// TwinCAT 3 PLC project MainPLCProject
// ProgramVersion: 3.1.4024.0
// libraries:
//   Tc2_Standard, * (Beckhoff Automation GmbH)
//   Tc2_System, * (Beckhoff Automation GmbH)
//   Tc2_TcpIp, * (Beckhoff Automation GmbH)
//   Tc2_Utilities, * (Beckhoff Automation GmbH)
//   Tc3_Module, * (Beckhoff Automation GmbH)
//   VisuDialogs, * (System)
//   VisuSymbols,3.5.10.0,System
// project tree:
//   DUTs/ ArmMovementState.TcDUT, ClientState.TcDUT, Command.TcDUT, COM_MODE.TcDUT, DataExchangeState.TcDUT, Message.TcDUT, MessageLogData.TcDUT, ReceiveStatus.TcDUT, SendStatus.TcDUT
//   DUTs/Robot Structs/ Joint.TcDUT, Position.TcDUT, RobotData.TcDUT, Timer.TcDUT
//   / GlobalTextList.TcGTLO, PlcTask.TcTTO, Visualization Manager.TcVMO (not stored)
//   GVLs/ GVL.TcGVL, GVL_Constants.TcGVL, GVL_RobotArmConstants.TcGVL
//   POUs/Classes/ ArmMovementHandler.TcPOU, COMMUNICATION.TcPOU, MESSAGE_CREATOR.TcPOU, MESSAGE_HANDLER.TcPOU, ROBOT_DATA_HANDLER.TcPOU, TCPClient.TcPOU
//   POUs/Helpers/ AddCounterToMessage.TcPOU, LogToWarning.TcPOU, ShiftHistoryLeft.TcPOU
//   POUs/InverseKinematics/ GetAngleDegreesFrom3Sides.TcPOU, GetAngleDegreesFromOppositeAndAdjacent.TcPOU, GetArm1AndArm2Degrees.TcPOU, GetArm3RotationPerpendicularToGround.TcPOU, GetBaseAngleDegrees.TcPOU, GetDistanceToPositionFromBase2D.TcPOU, GetHypotenuse.TcPOU, GetXSide.TcPOU, GetZSide.TcPOU, RadiansToDegrees.TcPOU
//   POUs/ MAIN.TcPOU
//   VISUs/ VisualizationControlPanel.TcVIS
// real-time tasks:
//   TASK PlcTask: cycle T#10ms, priority 20, ADS port 350
//   TASK HeartbeatTask: cycle T#50000us, priority 1, ADS port 351

CONFIGURATION MainPLCProject
    RESOURCE PLC ON TwinCAT3
        TASK PlcTask(INTERVAL := T#10ms, PRIORITY := 20);
        PROGRAM MAIN WITH PlcTask : MAIN;
    END_RESOURCE
END_CONFIGURATION

// ---- DUTs/ArmMovementState.TcDUT
{attribute 'qualified_only'}
{attribute 'strict'}
TYPE ArmMovementState :
(
	NONE,
	IDLE,
	PICKING,
	DROPPING
);
END_TYPE

// ---- DUTs/ClientState.TcDUT
{attribute 'qualified_only'}
{attribute 'strict'}
TYPE ClientState :
(
	IDLE,
	SENDING,
	RECEIVING
) := IDLE;
END_TYPE

// ---- DUTs/Command.TcDUT
TYPE Command :
STRUCT CONSTANT
	Start : STRING(9) := 'CRISTART';
	End : STRING(7) := 'CRIEND';
	MovementVar : STRING(4) := 'VAR';
	Heartbeat : STRING(9) := 'ALIVEJOG';
	
END_STRUCT
END_TYPE

// ---- DUTs/COM_MODE.TcDUT
{attribute 'qualified_only'}
{attribute 'strict'}
TYPE COM_MODE :
(
	Robot,
	Monarco
);
END_TYPE

// ---- DUTs/DataExchangeState.TcDUT
{attribute 'qualified_only'}
{attribute 'strict'}
TYPE DataExchangeState :
(
	IDLE,
	START,
	WORKING,
	ERROR
) := START;
END_TYPE

// ---- DUTs/Message.TcDUT
// Pre-made robot messages
TYPE Message :
STRUCT CONSTANT
	Connect : STRING(30) := 'CMD Connect';
	AliveDemo : STRING(63) := 'ALIVEJOG 40.0 50.0 40.0 30.0 30.0 0.0 0.0 0.0 0.0';	//Do not use, only for testing!
	EnableMessage : STRING(80) := 'CMD Enable';
END_STRUCT
END_TYPE

// ---- DUTs/MessageLogData.TcDUT
TYPE MessageLogData :
STRUCT
	systemTimeString : T_MaxString := '';
	message : STRING(GVL_Constants.MAX_RECEIVE_MESSAGE_LENGTH) := '';
END_STRUCT
END_TYPE

// ---- DUTs/ReceiveStatus.TcDUT
{attribute 'qualified_only'}
{attribute 'strict'}
TYPE ReceiveStatus :
(
	WAITING,
	RECEIVING,
	DONE,
	FAIL,
	TIMEOUT
) := RECEIVING;
END_TYPE

// ---- DUTs/Robot Structs/Joint.TcDUT
TYPE Joint :
STRUCT
	curPosition : LREAL;
	curSpeed : LREAL;
	setSpeed : LREAL;
	timer : TIMER;
END_STRUCT
END_TYPE

// ---- DUTs/Robot Structs/Position.TcDUT
TYPE Position :
STRUCT
	x : LREAL;	//Depth
	z : LREAL;	//Width
	y : LREAL;	//Height
END_STRUCT
END_TYPE

// ---- DUTs/Robot Structs/RobotData.TcDUT
TYPE RobotData :
STRUCT
	//Variables will be manipulated by Unity via ADS
	targetX : LREAL;
	targetY : LREAL;
	targetZ : LREAL;	
	isBusy : ARRAY[0..4] OF BOOL;	//Global value for all joints
	
	hasNewData : BOOL := FALSE;
	isAtDefaultPosition : BOOL := FALSE;	
	isAtDefaultPositionInt : INT := 0;		
	hasPickedUp : INT	:= 0;
	
	joint0 : Joint;
	joint1 : Joint;
	joint2 : Joint;
	joint3 : Joint;
	joint4 : Joint;
	
	
END_STRUCT
END_TYPE

// ---- DUTs/Robot Structs/Timer.TcDUT
TYPE Timer :
STRUCT
	timerTime : TIME;
	timerStart : BOOL;
	timerCon : TON;
END_STRUCT
END_TYPE

// ---- DUTs/SendStatus.TcDUT
{attribute 'qualified_only'}
{attribute 'strict'}
TYPE SendStatus :
(
	SENDING,
	FAIL,
	SUCCESS
) := SENDING;
END_TYPE

// ---- GVLs/GVL.TcGVL
{attribute 'qualified_only'}
VAR_GLOBAL
	// COMMUNICATION variables
	ReceivedStringArray : ARRAY[0..200] OF STRING;
	ReceivedStringWordCounter : INT := 0;

	ReceivedCMD : STRING := '';
	VarValue : STRING := '';
	VarType : STRING := '';
	VarName : STRING := '';
	//
	
	robotData : RobotData;
END_VAR

// ---- GVLs/GVL_Constants.TcGVL
{attribute 'qualified_only'}
VAR_GLOBAL CONSTANT
	MAX_RECEIVE_MESSAGE_LENGTH : UDINT := 2048;
	MAX_HISTORY_SIZE : BYTE := 10;
END_VAR

// ---- GVLs/GVL_RobotArmConstants.TcGVL
{attribute 'qualified_only'}
VAR_GLOBAL CONSTANT
	//All robot values are in mm
	PICKUP_AREA_DEPTH : LREAL := 60.0 * 10;
	PICKUP_AREA_WIDTH : LREAL := 60.0 * 10;
	
	//Values in mm
	DISTANCE_TO_PICKUP_AREA : LREAL := 90.0;	//Real: 90mm
	ARM_BASE_HEIGHT : LREAL := 310;
	GRABBER_HEIGHT : LREAL := 0.0;
	ARM_1_LENGTH : LREAL := 340.0;
	ARM_2_LENGTH : LREAL := 265.0;
	ARM_3_LENGTH : LREAL := 170.0;
	Pi : LREAL := 3.141592653589793238463;
	
	DROPOFF_X : LREAL := 450.0;	//MM	//TODO: Use DEPTH/2
	DROPOFF_Z : LREAL := PICKUP_AREA_WIDTH / 2;	//MM
	//Height is taken from the pickedup target
	DROPOFF_BASE_OFFSET : LREAL := -90.0;	//Degrees
	

	
	//Values in degrees
	MAXIMUM_BASE_ROTATION_FROM_CENTER : LREAL := 120.0;
	
END_VAR

// ---- POUs/MAIN.TcPOU
PROGRAM MAIN
VAR CONSTANT
	LOCAL_IP : T_IPv4Addr := '127.0.0.1';
	LOCAL_PORT : UDINT := 8080;

	REMOTE_IP : T_IPv4Addr := '192.168.3.1';
	REMOTE_PORT : UDINT := 8080;
	
	ROBOT_IP : T_IPv4Addr := '192.168.3.11';
	ROBOT_PORT : UDINT := 3920;
	
	MONARCO_IP : T_IPv4Addr := '192.168.3.125';
	MONARCO_PORT : UDINT := 8080;
	//TODO: Remove? not used anywhere afaik
	command : Command := ();
	message : Message := ();

	testPosition : Position := (x := 250.0, z := 250.0, y := 250.0);
	
END_VAR
VAR
	isSetUp : BOOL := FALSE;	

	buttonConnectPressed : BOOL;
	buttonDisconnectPressed : BOOL;	
	buttonSendPressed : BOOL;
	buttonConnectToRobotPressed : BOOL;
	buttonDebugSendPressed : BOOL;
	buttonEnableMotorsPressed : BOOL;
	buttonDisableMotorsPressed : BOOL;
	buttonLeft0Pressed : BOOL;
	buttonRight0Pressed : BOOL;
	buttonLeft1Pressed : BOOL;
	buttonRight1Pressed : BOOL;
	buttonLeft2Pressed : BOOL;
	buttonRight2Pressed : BOOL;
	buttonLeft3Pressed : BOOL;
	buttonRight3Pressed : BOOL;
	buttonStopPressed : BOOL;
	
	connectTrigger : R_TRIG;
	disconnectTrigger : R_TRIG;
	sendTrigger : R_TRIG;
	connectToRobotTrigger : R_TRIG;
	debugSendTrigger : R_TRIG;
	enableMotorsTrigger : R_TRIG;
	disableMotorsTrigger : R_TRIG;
	stopTrigger : R_TRIG;
	right0Trigger : R_TRIG;
	left0Trigger : R_TRIG;
	right1Trigger : R_TRIG;
	left1Trigger : R_TRIG;
	right2Trigger : R_TRIG;
	left2Trigger : R_TRIG;
	right3Trigger : R_TRIG;
	left3Trigger : R_TRIG;
	
	client : TCPClient(MONARCO_IP, MONARCO_PORT, isEnabled := FALSE);	//Note: make sure the COM_MODE is set properly, as it overwrites these values
	LocalSystemTime : FB_LocalSystemTime;
	
	// COMMUNICATION message handling
	MessageBase : COMMUNICATION(CommunicationMODE := COM_MODE.Robot); // change this to switch between robot and monarco mode!!
	messageHandler : MESSAGE_HANDLER();
	MessageERROR : int := 0;
	//
	// ROBOT_DATA handling
	RobotDataHandler : ROBOT_DATA_HANDLER;
	armMovementHandler : ArmMovementHandler;
	//
	
	connectionMessage : STRING(20) := 'Disconnected';
	isHeartbeatEnabled : BOOL := FALSE;
	
	closeAllConnections : FB_SocketCloseALL();
	closeAll : BOOL := TRUE;	//Close all on initial startup
	
	//messageToServer : T_MaxString := 'CRISTART 1 CMD Connect CRIEND';
	messageToServer : T_MaxString := 'Hello world 2.0 CRIEND';
	debugMessageToServer : T_MaxString := 'VAR Joint 0.0 0.0 0.0 0.0 0.0 0.0 0.0 0.0 0.0';
	messageFromServer : STRING(GVL_Constants.MAX_RECEIVE_MESSAGE_LENGTH) := '';
	//finalSendMsg : STRING(100);
	
	heartbeatTimer : TON;
	heartbeatInterval : TIME := T#100MS;
	
	sendCounter : INT := 1;
	finalAliveMessage : STRING(100) := '';
	totalMessagesFromServerCount : UDINT := 0;
	
	currentTime : TIMESTRUCT;
	messageHistoryArray : ARRAY [0.. GVL_Constants.MAX_HISTORY_SIZE - 1] OF MessageLogData;
	currentHistoryIndex : BYTE := 0;
	currentMessageLogData : MessageLogData;
	
	//Testing
	dummyHeartbeatValues : STRING(80);
	dummyMoveValues : STRING(80);
	

END_VAR

//On PLC reset/program download, close all connections
HandlePLCReset();

HandleSetup();
// === ===

// === UI Handling ===
HandleUI();

// === Message Sending ===
HandleMessageSending();

// === Message Handling ===
HandleMessageReceiving();

// === Heartbeat ===
HandleHeartbeat();

// === Arm movement ===
armMovementHandler();

// === Socket client ====
client(totalMessagesReceived => totalMessagesFromServerCount);



IF (GVL.robotData.isAtDefaultPosition = TRUE) THEN
	GVL.robotData.isAtDefaultPositionInt := 1;
ELSE
	GVL.robotData.isAtDefaultPositionInt := 0;
	
END_IF

METHOD PRIVATE HandleHeartbeat : BOOL
VAR_INPUT
END_VAR
heartbeatTimer(IN := isHeartbeatEnabled, PT := heartbeatInterval);

IF (heartbeatTimer.Q AND client.IsClientEnabled) THEN
	heartbeatTimer(IN := FALSE);
	// Send all movement data to the robot via the hardbeat.
	client.Send(messageToSend := MessageBase.CREATE('ALIVEJOG', RobotDataHandler.DATA_TO_STRING(), ERROR => MessageERROR));
END_IF
END_METHOD

METHOD PRIVATE HandleMessageReceiving : BOOL
VAR_INPUT
END_VAR
IF (client.NewMessageAvailable(clearFlag := TRUE)) THEN
	//Update history
	IF (currentHistoryIndex >= GVL_Constants.MAX_HISTORY_SIZE) THEN
		//Ran out of history space, discard youngest member
		currentHistoryIndex := GVL_Constants.MAX_HISTORY_SIZE;
		ShiftHistoryLeft(arr := messageHistoryArray);
	ELSE
		//Can still append
		currentHistoryIndex := currentHistoryIndex + 1;
	END_IF
	
	//Handle message
	MessageBase.HANDLE(messageFromServer);
	
	//Add new entry
	currentMessageLogData.message := messageFromServer;	
	currentMessageLogData.systemTimeString := SYSTEMTIME_TO_STRING(in := currentTime);
	messageHistoryArray[currentHistoryIndex - 1] := currentMessageLogData;
END_IF
END_METHOD

METHOD PRIVATE HandleMessageSending : BOOL
VAR_INPUT
END_VAR
CASE MessageBase.COMMUNICATION_MODE OF
	COM_MODE.Robot:
// ROBOT COM
		IF (sendTrigger.Q) THEN  // debug: send move command to robot.
			//TODO: Rework to use +- buttons (like in the C# application)
//			client.Send(messageToSend := MessageBase.CREATE(COMMAND := 'VAR', COMMAND_DETAILS := 'GetPosVariable Joint', ERROR => MessageERROR));
//			RobotDataHandler.DEGREES_TO_MOVEMENT_DATA(degrees := -45, jointNr := 0);
//			RobotDataHandler.DEGREES_TO_MOVEMENT_DATA(degrees := -34.8529, jointNr := 1);
//			RobotDataHandler.DEGREES_TO_MOVEMENT_DATA(degrees := -18.5157, jointNr := 2);
//			RobotDataHandler.DEGREES_TO_MOVEMENT_DATA(degrees := 53.3685, jointNr := 3);
			//RobotDataHandler.SET_JOINTS_TO_POSITION(X := 250.0, Z:= 250.0, Y := 250.0, baseOffsetDegrees := 0.0);
			
			GVL.robotData.targetX := 253.0;
			GVL.robotData.targetZ := 171.0;
			GVL.robotData.targetY := 160.0;
			
			GVL.robotData.hasNewData := TRUE;
		END_IF

		IF (debugSendTrigger.Q) THEN // debug: not in use yet.
//			client.Send(messageToSend := MessageBase.CREATE(COMMAND := 'CMD', COMMAND_DETAILS := 'Reset', ERROR => MessageERROR));
			RobotDataHandler.DEGREES_TO_MOVEMENT_DATA(degrees := 0, jointNr := 0);
			RobotDataHandler.DEGREES_TO_MOVEMENT_DATA(degrees := 0, jointNr := 1);
			RobotDataHandler.DEGREES_TO_MOVEMENT_DATA(degrees := 0, jointNr := 2);
			RobotDataHandler.DEGREES_TO_MOVEMENT_DATA(degrees := 0, jointNr := 3);
		END_IF
		
		IF (left0Trigger.Q) THEN  // debug: send move command to robot.
			GVL.robotData.joint0.curSpeed := 20.0;
		END_IF
		
		IF (right0Trigger.Q) THEN 
			
			GVL.robotData.joint0.curSpeed := -20.0;
		END_IF
		
		IF (left1Trigger.Q) THEN  // debug: send move command to robot.
			GVL.robotData.joint1.curSpeed := 20.0;
		END_IF
		
		IF (right1Trigger.Q) THEN 
			
			GVL.robotData.joint1.curSpeed := -20.0;
		END_IF
		
		IF (left2Trigger.Q) THEN  // debug: send move command to robot.
			GVL.robotData.joint2.curSpeed := 20.0;
		END_IF
		
		IF (right2Trigger.Q) THEN 
			
			GVL.robotData.joint2.curSpeed := -20.0;
		END_IF
		
		IF (left3Trigger.Q) THEN  // debug: send move command to robot.
			GVL.robotData.joint3.curSpeed := 20.0;
		END_IF
		
		IF (right3Trigger.Q) THEN 
			
			GVL.robotData.joint3.curSpeed := -20.0;
		END_IF
		
		IF (stopTrigger.Q) THEN 
			GVL.robotData.joint0.curSpeed := 0.0;
			GVL.robotData.joint1.curSpeed := 0.0;
			GVL.robotData.joint2.curSpeed := 0.0;
			GVL.robotData.joint3.curSpeed := 0.0;
		END_IF

		IF (connectToRobotTrigger.Q) THEN
			client.Send(messageToSend := MessageBase.CREATE(COMMAND := 'CMD', COMMAND_DETAILS := 'Connect', ERROR => MessageERROR));
			isHeartbeatEnabled := TRUE;
		END_IF

		IF (enableMotorsTrigger.Q) THEN
			client.Send(messageToSend := MessageBase.CREATE(COMMAND := 'CMD', COMMAND_DETAILS := 'Enable', ERROR => MessageERROR));
		END_IF
		
		IF (disableMotorsTrigger.Q) THEN
			client.Send(messageToSend := MessageBase.CREATE(COMMAND := 'CMD', COMMAND_DETAILS := 'Disable', ERROR => MessageERROR));
		END_IF
//		
	COM_MODE.Monarco:
// MONARCO COM
		IF (sendTrigger.Q) THEN 
			client.Send(messageToSend := MessageBase.CREATE(COMMAND := 'CMD', COMMAND_DETAILS := 'LED_ON', ERROR => MessageERROR));
		END_IF

		IF (debugSendTrigger.Q) THEN
			client.Send(messageToSend := MessageBase.CREATE(COMMAND := 'CMD', COMMAND_DETAILS := 'LED_OFF', ERROR => MessageERROR));
		END_IF
//
END_CASE
END_METHOD

METHOD HandlePLCReset : BOOL
VAR_INPUT
END_VAR
IF (closeAll) THEN	
	closeAll := FALSE;
	closeAllConnections(sSrvNetId := '', bExecute := TRUE, tTimeout := T#10S);
ELSE
	closeAllConnections(bExecute := FALSE);
END_IF

IF (closeAllConnections.bBusy) THEN
	RETURN;	//Do not continue the program until all connections are closed
END_IF
END_METHOD

METHOD HandleSetup : BOOL
VAR_INPUT
END_VAR
IF (NOT isSetUp) THEN
	armMovementHandler.BindRobotDataHandler(dataHandler := RobotDataHandler);

	isSetUp := TRUE;
END_IF
END_METHOD

METHOD HandleUI : BOOL
VAR_INPUT
END_VAR
LocalSystemTime(bEnable := TRUE, tTimeout := T#1S, systemTime => currentTime);

connectTrigger(CLK := buttonConnectPressed);
disconnectTrigger(CLK := buttonDisconnectPressed);
sendTrigger(CLK := buttonSendPressed);
connectToRobotTrigger(CLK := buttonConnectToRobotPressed);
debugSendTrigger(CLK := buttonDebugSendPressed);
enableMotorsTrigger(CLK := buttonEnableMotorsPressed);
disableMotorsTrigger(CLK := buttonDisableMotorsPressed);
left0Trigger(CLK := buttonLeft0Pressed);
right0Trigger(CLK := buttonRight0Pressed);
left1Trigger(CLK := buttonLeft1Pressed);
right1Trigger(CLK := buttonRight1Pressed);
left2Trigger(CLK := buttonLeft2Pressed);
right2Trigger(CLK := buttonRight2Pressed);
left3Trigger(CLK := buttonLeft3Pressed);
right3Trigger(CLK := buttonRight3Pressed);
stopTrigger(CLK := buttonStopPressed);

IF (client.IsConnected) THEN
	connectionMessage := 'Connected';
ELSE
	connectionMessage := 'Disconnected';
END_IF

IF (connectTrigger.Q) THEN
	//Note: Not sure if this is a good idea, as it is burried in the code and can lead to unexpected behaviour
	CASE MessageBase.COMMUNICATION_MODE OF
	// check for communication mode and set IP for this mode.
		COM_MODE.Robot:
			client.RemoteServerAddress := ROBOT_IP;
			client.RemoteServerPort := ROBOT_PORT;
		
		COM_MODE.Monarco:
			client.RemoteServerAddress := MONARCO_IP;
			client.RemoteServerPort := MONARCO_PORT;
	END_CASE
	client.BindReceiveMessage(variableToBind := messageFromServer);
	client.Enable();
END_IF

IF (disconnectTrigger.Q) THEN
	client.Disable();
END_IF
END_METHOD

END_PROGRAM

// ---- POUs/Classes/TCPClient.TcPOU
FUNCTION_BLOCK TCPClient
VAR CONSTANT
	CLIENT_RECONNECT_TIME : TIME := T#31S;
	MAX_MESSAGE_LENGTH : INT := 255;
	MAX_RECEIVE_MESSAGE_LENGTH : UDINT := GVL_Constants.MAX_RECEIVE_MESSAGE_LENGTH;
END_VAR
VAR_OUTPUT
	totalMessagesReceived : UDINT := 0;
END_VAR
VAR
	m_isClientEnabled : BOOL := TRUE;	
	m_serverNetID : STRING(80) := '';
	
	ClientServerConnection : FB_ClientServerConnection;
	SocketSend : FB_SocketSend;
	SocketReceive : FB_SocketReceive;
	//m_clientDataExchanger : ClientDataExchanger;	//Note implemented yet: leave for later, use as
	m_socketHandle : T_HSOCKET;
	
	
	m_remoteServerAddress : T_IPv4Addr;	
	m_remoteServerPort : UDINT := 0;
	
	//Note: make it an input and send only when the class is called?
	m_messageToSend : T_MaxString := 'Hello world!';
	//m_messageReceived : T_MaxString;	// The latest message received from the server //TODO: REMOVE, Depricated
	m_messageReceivedRef : REFERENCE TO STRING(MAX_RECEIVE_MESSAGE_LENGTH);
	
	m_isConnected : BOOL := FALSE;
	m_isBusy : BOOL;
	m_errorOccured : BOOL;
	m_lastErrorId : UDINT;
	
	
	m_currentSocketState : Tc2_TcpIp.E_SocketConnectionState;
	m_currentState : ClientState := ClientState.RECEIVING;	

	m_sendDataExchangeState : DataExchangeState := DataExchangeState.START;	
	m_sendRequested: BOOL;
	m_sendStatus : SendStatus;
	m_sendErrorId : UDINT;
	m_sendTimeout : TIME := T#15S;	//Note: Lower?
	//m_sendTimeout : TIME := T#1M;	//Note: Lower?
	
	//Receiving
	m_receiveDataExchangeState : DataExchangeState := DataExchangeState.IDLE;	
	m_isReceiveTimerEnabled : BOOL := TRUE;
	m_receiveTimer : TON();
	m_isReceiveTimeoutEnabled : BOOL := FALSE;	
	m_receiveTimeoutTimer : TON();
	m_receiveBuffer : STRING(MAX_RECEIVE_MESSAGE_LENGTH) := '';
	m_totalBytesReceived : UDINT := 0;
	m_receiveTimeout : TIME := T#1M;
	m_readInterval : TIME := T#10MS;
//	m_receiveMessageDelimiter : BYTE := F_ToASC(';');	//Note: Use plain 0 (without F_ToASC()) for \0
	m_receiveMessageDelimiter : BYTE := 0;	//'\0'	//Not used currently
	m_delimiterString : STRING(80) := 'CRIEND';
	m_receivedMessage : T_MaxString := '';
	m_receiveStatus : ReceiveStatus;
	m_newDataAvailable : BOOL := FALSE;	//Reset to false when it is read
	m_receiveErrorId : UDINT := 0;
	m_totalMessagesReceived : UDINT := 0;
END_VAR

//Handler code
//Does that need to be executed every cycle or can I put it in eSOCKET_DISCONNECTED state?
ClientServerConnection(sSrvNetID := m_serverNetID,
						 nMode := 0,
						 sRemoteHost := RemoteServerAddress,
						 nRemotePort := m_remoteServerPort,
						 tReconnect := CLIENT_RECONNECT_TIME,	//MAYBE
						 bEnable := IsClientEnabled,
						 bBusy => m_isBusy,
						 bError => m_errorOccured,
						 nErrId => m_lastErrorId,
						 hSocket => m_socketHandle,
						 eState => m_currentSocketState);

CASE m_currentSocketState OF
	E_SocketConnectionState.eSOCKET_DISCONNECTED:
		m_isConnected := FALSE;
	//
	E_SocketConnectionState.eSOCKET_SUSPENDED:
	//Change from disconnected to connected or vise versa
		m_isConnected := FALSE;
	//
	E_SocketConnectionState.eSOCKET_CONNECTED:
		m_isConnected := TRUE;
END_CASE

IF (NOT m_isConnected) THEN
	RETURN;
END_IF

// Executed only if a connection is established

CASE m_currentState OF
	//
	ClientState.SENDING:
		m_sendStatus := SendMessage(messageToSend := m_messageToSend, timeout := m_sendTimeout, errorId => m_sendErrorId);
		IF (m_sendStatus = SendStatus.SUCCESS) THEN
			m_currentState := ClientState.RECEIVING;
		ELSIF (m_sendStatus = SendStatus.FAIL) THEN
			//Sending failed
			ADSLOGDINT(msgCtrlMask := ADSLOG_MSGTYPE_WARN, msgFmtStr := 'Send fail error: %d', dintArg := UDINT_TO_DINT(m_sendErrorId));
			m_currentState := ClientState.RECEIVING;
		END_IF
		
	//
	ClientState.RECEIVING:
		m_receiveStatus := Receive(timeout := m_receiveTimeout, 
									readInterval := m_readInterval, 
									messageDelimiter := m_receiveMessageDelimiter,	//Currently not used
									errorId => m_receiveErrorId);
		
		IF (m_receiveStatus <> ReceiveStatus.RECEIVING) THEN
			IF (m_receiveStatus = ReceiveStatus.DONE) THEN
				//
				totalMessagesReceived := totalMessagesReceived + 1;
				m_newDataAvailable := TRUE;
			END_IF
			
			IF (m_receiveStatus = ReceiveStatus.FAIL) THEN
				//Fail Handling
				//How does it get to error and the error is 0??
				LogToWarning(msgFmtStr := 'Receive fail error: %s', messageArg := UDINT_TO_STRING(m_receiveErrorId));
			END_IF
			
			IF (m_receiveStatus = ReceiveStatus.TIMEOUT) THEN
				//Timeout handling
				LogToWarning(msgFmtStr := 'Receive timed out', messageArg := '');
				//Disable();	//Disable on timeout
			END_IF
	
			IF (m_sendRequested) THEN
				m_sendRequested := FALSE;
				m_sendErrorId := 0;
				m_currentState := ClientState.SENDING;
			END_IF
		END_IF						
	
	// After done receiving, go to idle?
	//
END_CASE

METHOD PUBLIC BindReceiveMessage : BOOL
VAR_INPUT
	variableToBind : REFERENCE TO STRING(MAX_RECEIVE_MESSAGE_LENGTH);
END_VAR
m_messageReceivedRef REF= variableToBind;
END_METHOD

METHOD PUBLIC Disable : BOOL
m_isClientEnabled := False;
END_METHOD

METHOD PUBLIC Enable : BOOL
VAR_INPUT
END_VAR
m_isClientEnabled := TRUE;
END_METHOD

METHOD FB_init : BOOL
VAR_INPUT
	bInitRetains : BOOL; // if TRUE, the retain variables are initialized (warm start / cold start)
	bInCopyCode : BOOL;  // if TRUE, the instance afterwards gets moved into the copy code (online change)
	
	remoteServerAddress : T_IPv4Addr := '127.0.0.1';
	remoteServerPort : UDINT := 8080;
	isEnabled : BOOL := FALSE;
END_VAR
m_remoteServerAddress := remoteServerAddress;
m_remoteServerPort := remoteServerPort;
m_isClientEnabled := isEnabled;
END_METHOD

PROPERTY IsClientEnabled : BOOL
GET
IsClientEnabled := m_isClientEnabled;
END_GET
END_PROPERTY

PROPERTY IsConnected : BOOL
GET
IsConnected := m_isConnected;
END_GET
END_PROPERTY

PROPERTY LastSendStatus : SendStatus
GET
LastSendStatus := m_sendStatus;
END_GET
END_PROPERTY

METHOD PUBLIC NewMessageAvailable : BOOL
VAR_INPUT
	clearFlag : BOOL := FALSE;	//Clears the new message flag if set to true, does not otherwise
END_VAR
NewMessageAvailable := m_newDataAvailable;

IF (clearFLag) THEN
	m_newDataAvailable := FALSE;
END_IF
END_METHOD

METHOD PRIVATE Receive : ReceiveStatus
VAR_INPUT
	timeout : TIME;// := T#10S;
	readInterval : TIME := T#10MS;
	messageDelimiter : BYTE := 0;
END_VAR

VAR_OUTPUT
	errorId : UDINT;
END_VAR

VAR
	errorOccurred : BOOL;	//can sty
	isBusy : BOOL;	//can stay																
	
	timedout : BOOL := FALSE;	//Output of TON
	receivedBytes : UDINT := 0;	//Output, should be fine to be here
	
	startPosition : UDINT := 0;	//Can stay, assigned before used
	endPosition : UDINT := 0;	//Can stay, assigned before used
	currentFrameLength : UDINT := 0; // Length of string received this cycle	//Should be fine
	posOfDelimiter : UDINT := 0;
	
	
	index : UDINT := 0;	//For-loop index
	
END_VAR
m_receiveTimer(IN := m_isReceiveTimerEnabled);
m_receiveTimeoutTimer(IN := m_isReceiveTimeoutEnabled, PT := timeout, Q => timedout);

CASE m_receiveDataExchangeState OF
	DataExchangeState.IDLE:
		//Reset variables
		m_isReceiveTimerEnabled := FALSE;
		m_receiveTimer(IN := m_isReceiveTimerEnabled, PT := T#0MS); 	//Do not wait for the first read
		m_isReceiveTimeoutEnabled := FALSE;
		Receive := ReceiveStatus.WAITING;
		m_receiveDataExchangeState := DataExchangeState.START;
	//
	DataExchangeState.START:
		Receive := ReceiveStatus.WAITING;
		m_isReceiveTimerEnabled := TRUE;
		IF (m_receiveTimer.Q) THEN
			SocketReceive(bExecute := FALSE);
			SocketReceive(sSrvNetId := m_serverNetID,
						  hSocket := m_socketHandle,
						  pDest := ADR(m_receiveBuffer) + m_totalBytesReceived,
						  cbLen := SIZEOF(m_receiveBuffer) - m_totalBytesReceived,
						  tTimeout := timeout,
						  bExecute := TRUE);	
			
			m_receiveDataExchangeState := DataExchangeState.WORKING;
		END_IF
	//
	DataExchangeState.WORKING:
		Receive := ReceiveStatus.RECEIVING;
		SocketReceive(bExecute := FALSE,
				tTimeout := timeout,
				bBusy => isBusy,
				bError => errorOccurred,
				nErrId => errorId,
				nRecBytes => receivedBytes);
		//Enable timeout
		IF (NOT isBusy AND NOT errorOccurred) THEN
			IF (receivedBytes > 0) THEN
				startPosition := m_totalBytesReceived;
				//Calculate new total
				m_totalBytesReceived := m_totalBytesReceived + receivedBytes;
				endPosition := m_totalBytesReceived - 1;
				currentFrameLength := 0;
				//Only proceed if we have enough space
				IF (m_totalBytesReceived < SIZEOF(m_messageReceivedRef)) THEN
					m_receiveTimer (PT := T#0MS); //Read asap
					//Bytes received, disable timeout check
					m_isReceiveTimeoutEnabled := FALSE;
					//Search for end of message delimiter
					
					posOfDelimiter := INT_TO_UDINT(FIND(STR1 := m_receiveBuffer, STR2 := m_delimiterString));
					
					IF (posOfDelimiter = 0) THEN
						//Delimiter not found
						LogToWarning('Delim not found', '');
						RETURN;
					END_IF
					
					currentFrameLength := posOfDelimiter + 6(*delimiter size*);
					//reset dest
					m_messageReceivedRef := '';
					MEMCPY(destAddr := ADR(m_messageReceivedRef), srcAddr := ADR(m_receiveBuffer), n := currentFrameLength);
					MEMSET(destAddr := ADR(m_receiveBuffer), fillByte := 0, n := SIZEOF(m_receiveBuffer));	//Clear buffer
					m_totalBytesReceived := 0;
					
					//All received
					Receive := ReceiveStatus.DONE;
					m_receiveDataExchangeState := DataExchangeState.IDLE;
					(*
					//OLD Find TODO: Find a way to implement via a function? So that you can use both
					FOR index := startPosition TO endPosition BY 1 DO
						IF (m_receiveBuffer[index] = messageDelimiter) THEN	//End of message check
							//End of message received
							currentFrameLength := index + 1;
							
							MEMCPY(destAddr := ADR(m_messageReceivedRef), srcAddr := ADR(m_receiveBuffer), n := currentFrameLength);
							//Move the remaining data bytes to the begining
							MEMMOVE(ADR(m_receiveBuffer), ADR(m_receiveBuffer[currentFrameLength]), m_totalBytesReceived - currentFrameLength); 
							//Recalculate remaining data byte length
							m_totalBytesReceived := m_totalBytesReceived - currentFrameLength;
							//All received
							Receive := ReceiveStatus.DONE;
							m_receiveDataExchangeState := DataExchangeState.IDLE;
							EXIT;
						END_IF
					END_FOR
					*)
				ELSE	
					//No more space in the receive object
					Receive := ReceiveStatus.FAIL;
					errorId := 42;
					//LogToWarning('totalBytesReceived exceeded limit: Received: %s', UDINT_TO_STRING(receivedBytes));
					m_receiveDataExchangeState := DataExchangeState.ERROR;
				END_IF //IF (totalBytesReceived < SIZEOF(receivedMessage))
			ELSE
				//No bytes received
				m_receiveTimer (PT := readInterval);
				m_isReceiveTimeoutEnabled := TRUE;
				
				//IF (timedout) THEN
				IF (m_receiveTimeoutTimer.Q) THEN
					Receive := ReceiveStatus.TIMEOUT;
					m_receiveDataExchangeState := DataExchangeState.ERROR;
					LogToWarning('Timed out!', '');
				ELSE
					//Read again
					m_receiveDataExchangeState := DataExchangeState.START;
				END_IF
			END_IF //IF (receivedBytes > 0)
		
		ELSIF (errorOccurred) THEN
			Receive := ReceiveStatus.FAIL;
			m_receiveDataExchangeState := DataExchangeState.ERROR;
		END_IF	//IF (NOT isBusy AND NOT errorOccurred)
		
	//
	DataExchangeState.ERROR:
		//Variable resets in case of an error
		m_totalBytesReceived := 0;	//Reset counter
		m_receiveBuffer := DELETE(STR := m_receiveBuffer, POS := 1, LEN := 255);	//Reset receive buffer
		m_receiveDataExchangeState := DataExchangeState.IDLE;
	//
END_CASE
END_METHOD

//Note: After reading, NewDataAvailable returns false until new data arrives
PROPERTY ReceivedData : T_MaxString
GET
ReceivedData := m_receivedMessage;
m_newDataAvailable := FALSE;
END_GET
END_PROPERTY

PROPERTY RemoteServerAddress : T_IPv4Addr
GET
RemoteServerAddress := m_remoteServerAddress;
END_GET
SET
m_remoteServerAddress := RemoteServerAddress;
END_SET
END_PROPERTY

PROPERTY RemoteServerPort : UDINT
GET
RemoteServerPort := m_remoteServerPort;
END_GET
SET
m_remoteServerPort := RemoteServerPort;
END_SET
END_PROPERTY

METHOD Send : BOOL
VAR_INPUT
	messageToSend : T_MaxString;
END_VAR
m_sendRequested := TRUE;
m_messageToSend := messageToSend;
END_METHOD

//Wrapper for SocketSend. On error, check the errorId variable
METHOD PRIVATE SendMessage : SendStatus
VAR_INPUT
	messageToSend : T_MaxString;
	timeout : TIME;
END_VAR

VAR_OUTPUT
	errorId : UDINT := 0;
END_VAR

VAR
	errorOccurred : BOOL;	
	isBusy : BOOL;	
END_VAR
CASE m_sendDataExchangeState OF
	DataExchangeState.START:
		errorId := 0;
		
		SocketSend(sSrvNetId := m_serverNetID,
				   hSocket := m_socketHandle,
				   cbLen := INT_TO_UDINT(LEN(messageToSend) + 1),
		   		   pSrc := ADR(messageToSend),
				   tTimeout := timeout,
				   bExecute := FALSE
				   );

		m_sendDataExchangeState := DataExchangeState.WORKING;
	//
	DataExchangeState.WORKING:
		
		SocketSend(bExecute := TRUE,
				   bError => errorOccurred,
		   		   nErrId => errorId,
		   		   bBusy => isBusy);
		
		IF (NOT isBusy AND NOT errorOccurred) THEN
			SendMessage := SendStatus.SUCCESS;
			m_sendDataExchangeState := DataExchangeState.START;
		ELSIF (errorOccurred) THEN
			SendMessage := SendStatus.FAIL;
			m_sendDataExchangeState := DataExchangeState.START;
		ELSIF (isBusy) THEN
			SendMessage := SendStatus.SENDING;
		END_IF 
	//
END_CASE
END_METHOD

END_FUNCTION_BLOCK

// ---- POUs/Helpers/LogToWarning.TcPOU
FUNCTION LogToWarning : BOOL
VAR_INPUT
	msgFmtStr : T_MaxString;
	messageArg : T_MaxString;
END_VAR
VAR
END_VAR

ADSLOGSTR(msgCtrlMask := ADSLOG_MSGTYPE_WARN, msgFmtStr := msgFmtStr, strArg := messageArg);

END_FUNCTION

// ---- POUs/Classes/COMMUNICATION.TcPOU
FUNCTION_BLOCK COMMUNICATION
VAR_INPUT
	
END_VAR
VAR_OUTPUT
END_VAR
VAR
	m_COMMUNICATION_MODE : COM_MODE;
	messageCreator : MESSAGE_CREATOR('CRISTART', 'CRIEND', 1);
	messageHandler : MESSAGE_HANDLER();
END_VAR

PROPERTY PUBLIC COMMUNICATION_MODE : COM_MODE
GET
COMMUNICATION_MODE := m_COMMUNICATION_MODE;
END_GET
SET
m_COMMUNICATION_MODE := COMMUNICATION_MODE;
END_SET
END_PROPERTY

METHOD PUBLIC CREATE : STRING
VAR_INPUT
	COMMAND : STRING;
	COMMAND_DETAILS : STRING;
END_VAR
VAR_OUTPUT
	ERROR : INT := 0;
END_VAR
IF (COMMUNICATION_MODE = COM_MODE.Robot) THEN 
	// creates string for robot when in Robot mode
	CREATE := MessageCreator.ROBOT_MESSAGE(COMMAND, COMMAND_DETAILS, ERROR => ERROR);
ELSIF (COMMUNICATION_MODE = COM_MODE.Monarco) THEN 
	// creates string for monarco when in Monarco mode
	CREATE := MessageCreator.MONARCO_MESSAGE_CMD(COMMAND_DETAILS, ERROR => ERROR);
			// JUST THE CMD MONARCO MESSAGE FOR NOW!!
END_IF
END_METHOD

METHOD FB_init : BOOL
VAR_INPUT
	bInitRetains : BOOL; // if TRUE, the retain variables are initialized (warm start / cold start)
	bInCopyCode : BOOL;  // if TRUE, the instance afterwards gets moved into the copy code (online change)
	
	communicationMODE : COM_MODE;
END_VAR
COMMUNICATION_MODE := communicationMode;
END_METHOD

METHOD PUBLIC HANDLE : INT
VAR_INPUT
	FULL_STRING : STRING;
END_VAR
IF (COMMUNICATION_MODE = COM_MODE.Robot) THEN 
	// handles string from robot when in Robot mode (RECEIVE_ROBOT())
	MessageHandler.RECEIVE_ROBOT(FULL_STRING, ERROR => HANDLE);
ELSIF (COMMUNICATION_MODE = COM_MODE.Monarco) THEN 
	// handles string from monarco when in Monarco mode (RECEIVE_MONARCO())
	MessageHandler.RECEIVE_MONARCO(FULL_STRING, ERROR => HANDLE);
END_IF
END_METHOD

END_FUNCTION_BLOCK

// ---- POUs/Classes/MESSAGE_CREATOR.TcPOU
FUNCTION_BLOCK PUBLIC MESSAGE_CREATOR
VAR_INPUT
END_VAR
VAR_OUTPUT
END_VAR
VAR
	m_START_COMMAND : STRING;
	m_END_COMMAND : STRING;
	m_MESSAGE_COUNT : INT;
END_VAR

PROPERTY PUBLIC END_COMMAND : STRING
GET
END_COMMAND := m_END_COMMAND;
END_GET
SET
m_END_COMMAND := END_COMMAND;
END_SET
END_PROPERTY

METHOD FB_init : BOOL
VAR_INPUT
	bInitRetains : BOOL; // if TRUE, the retain variables are initialized (warm start / cold start)
	bInCopyCode : BOOL;  // if TRUE, the instance afterwards gets moved into the copy code (online change)
	
	STARTcommand : STRING;
	ENDcommand : STRING;
	MESSAGEcount : INT;
END_VAR
START_COMMAND := STARTcommand;
END_COMMAND := ENDcommand;
MESSAGE_COUNT := MESSAGEcount;
END_METHOD

PROPERTY PUBLIC MESSAGE_COUNT : INT
GET
MESSAGE_COUNT := m_MESSAGE_COUNT;
END_GET
SET
m_MESSAGE_COUNT := MESSAGE_COUNT;
END_SET
END_PROPERTY

METHOD PUBLIC MONARCO_MESSAGE_CMD : STRING
VAR_INPUT
	COMMAND_DETAILS : STRING;
END_VAR
VAR CONSTANT
	COMMAND : STRING := 'CMD';
	SEPARATOR : STRING := ' ';
END_VAR
VAR_OUTPUT
	ERROR : INT := 0;
END_VAR
IF (COMMAND_DETAILS <> '') THEN // if command_details is not empty, create command string.
	MONARCO_MESSAGE_CMD := 
		CONCAT(COMMAND, 
		CONCAT(SEPARATOR, 
			COMMAND_DETAILS));
			
ELSE // else return error string and error code 1.
	MONARCO_MESSAGE_CMD := 'ERROR_NoCommandDetailsGiven';
	ERROR := 1;
END_IF

//FULL_MONARCO_CMD_MESSAGE := 'CMD TURN_LED_ON';
END_METHOD

METHOD PUBLIC MONARCO_MESSAGE_VAR : STRING
VAR_INPUT
	VARIABLE_NAME : STRING;
	VARIABLE_TYPE : STRING;
	VARIABLE_VALUE : STRING;
END_VAR
VAR CONSTANT
	COMMAND : STRING := 'VAR';
	SEPARATOR : STRING := ' ';
END_VAR
VAR_OUTPUT
	ERROR : INT := 0;
END_VAR
IF (VARIABLE_NAME <> '' AND VARIABLE_TYPE <> '' AND VARIABLE_VALUE <> '') THEN 
	// if all values given, create var string.
	MONARCO_MESSAGE_VAR := 
			CONCAT(COMMAND, 
			CONCAT(SEPARATOR, 
			CONCAT(VARIABLE_NAME,
			CONCAT(SEPARATOR, 
			CONCAT(VARIABLE_TYPE,
			CONCAT(SEPARATOR, 
				VARIABLE_VALUE))))));
				
ELSE // else return error string, and error code 1.
	MONARCO_MESSAGE_VAR := 'ERROR_SomeValuesMissing';
	ERROR := 1;
END_IF

//FULL_MONARCO_VAR_MESSAGE := 'CMD varName1 INT 9';
END_METHOD

METHOD PUBLIC ROBOT_MESSAGE : T_MaxString
VAR_INPUT
	COMMAND : STRING;
	COMMAND_DETAILS : STRING;
END_VAR
VAR_OUTPUT
	ERROR : INT := 0;
END_VAR
 // CREATES A STRING THAT THE IGUS ROBOT CAN READ AND UNDERSTAND VIA ETHERNET.
ROBOT_MESSAGE := 
CONCAT(START_COMMAND, 
CONCAT(' ', 
CONCAT(INT_TO_STRING(MESSAGE_COUNT), 
CONCAT(' ', 
CONCAT(COMMAND, 
CONCAT(' ', 
CONCAT(COMMAND_DETAILS, 
CONCAT(' ', END_COMMAND))))))));

MESSAGE_COUNT := (MESSAGE_COUNT MOD 9999)+ 1;

//FULL_ROBOT_MESSAGE := 'CRISTART 1 CMD Connect CRIEND';
END_METHOD

PROPERTY PUBLIC START_COMMAND : STRING
GET
START_COMMAND := m_START_COMMAND;
END_GET
SET
m_START_COMMAND := START_COMMAND;
END_SET
END_PROPERTY

END_FUNCTION_BLOCK

// ---- POUs/Classes/MESSAGE_HANDLER.TcPOU
FUNCTION_BLOCK PUBLIC MESSAGE_HANDLER
VAR_INPUT
END_VAR
VAR_OUTPUT
END_VAR
VAR
END_VAR

METHOD FB_init : BOOL
VAR_INPUT
	bInitRetains : BOOL; // if TRUE, the retain variables are initialized (warm start / cold start)
	bInCopyCode : BOOL;  // if TRUE, the instance afterwards gets moved into the copy code (online change)

	
END_VAR
END_METHOD

METHOD PUBLIC RECEIVE_MONARCO : INT
VAR_INPUT
	FULL_STRING : STRING;
END_VAR
VAR
	FOUND_SEPARATOR : BOOL;
	COMMAND_CMD : STRING := 'CMD';
	COMMAND_VAR : STRING := 'VAR';
	count : INT := 0;
	MESSAGE_ARRAY : ARRAY[1..4] OF STRING;
	
	SeparatorChar : STRING := ' ';
	tempString : STRING := '';
	stringLeft : STRING := '';
	stringLeftSize : UDINT := 999;
	stringRight : STRING := '';
	stringRightSize : UDINT := 999;
END_VAR
VAR_OUTPUT
	ERROR : INT := 0;
END_VAR
// save received string into changeble variable.

tempString := FULL_STRING;

FOR count := 1 TO 4 BY 1 DO
	FOUND_SEPARATOR := FindAndSplitChar(
		sSeparatorChar := SeparatorChar, 	// split when this char found
		pSrcString := ADR(tempString), 		// string that will be split
		pLeftString := ADR(stringLeft), 	// first string (left) (FIRST WORD)
		nLeftSize := stringLeftSize, 		// first string size (right)
		pRightString := ADR(stringRight), 	// second string (right) (REST OF STRING)
		nRightSize := stringRightSize, 		// second string size (right)
		bSearchFromright := FALSE);			// when false start searching from the left
		
	IF FOUND_SEPARATOR THEN
		MESSAGE_ARRAY[count] := stringLeft; // saving the left string in message_array.
		tempString := stringRight; // saving the rest of the string for the next split.
	ELSE // ERROR: the separator char could not be found.
		MESSAGE_ARRAY[count] := tempString; // saving the string in case it was the last word.
		ERROR := count; 
		count := 10;
	END_IF
END_FOR

IF (ERROR = 2 OR ERROR = 4) THEN // handle message_array when CMD or VAR was the command.
	ERROR := 0;
	IF (MESSAGE_ARRAY[1] = COMMAND_CMD) THEN // when CMD was the command.
		GVL.ReceivedCMD := MESSAGE_ARRAY[2];
	ELSIF (MESSAGE_ARRAY[1] = COMMAND_VAR) THEN // when VAR was the command.
		GVL.VarName := MESSAGE_ARRAY[2];
		GVL.VarType := MESSAGE_ARRAY[3];
		GVL.VarValue := MESSAGE_ARRAY[4];
	ELSE
		ERROR := 5; // ERROR: neither CMD or VAR was red.
	END_IF
END_IF
END_METHOD

METHOD PUBLIC RECEIVE_ROBOT : INT
VAR_INPUT
	FULL_STRING : STRING;
END_VAR
VAR
	tempString : STRING;
	SeparatorChar : STRING := ' ';
	stringLeft : STRING;
	stringLeftSize : UDINT := 999;
	stringRight : STRING;
	stringRightSize : UDINT := 999;
	foundSeparator : BOOL;
	
	stepCount : INT;
END_VAR
VAR_OUTPUT
	ERROR : INT;
END_VAR
tempString := FULL_STRING;
FOR stepCount := 0 TO 200 BY 1 DO
	foundSeparator := FindAndSplitChar( // SEPERATE THE STRING, FIRST WORD -- REST OF STRING
		sSeparatorChar := SeparatorChar, 	// split when this char found
		pSrcString := ADR(tempString), 		// string that will be split
		pLeftString := ADR(stringLeft), 	// first string (left) (FIRST WORD)
		nLeftSize := stringLeftSize, 		// first string size (right)
		pRightString := ADR(stringRight), 	// second string (right) (REST OF STRING)
		nRightSize := stringRightSize, 		// second string size (right)
		bSearchFromright := FALSE);			// when false start searching from the left
	IF (stringRight = 'CRIEND') THEN // CHECK FOR ENDING
		GVL.ReceivedStringArray[stepCount] := stringLeft;
		GVL.ReceivedStringArray[stepCount + 1] := stringRight;
		GVL.ReceivedStringWordCounter := (stepCount + 1);
		stepCount := 210;
		ERROR := 0;
	ELSE // OTHERWISE SAVE SEPPERATED VAR AND CONTINUE
		IF (foundSeparator) THEN // CHECK FOR ERROR
			tempString := stringRight;
			GVL.ReceivedStringArray[stepCount] := stringLeft;
		ELSE // ERROR OCCURED, COULD NOT FIND SEPARATOR
			stepCount := 210;
			ERROR := 3;
		END_IF 
	END_IF 
END_FOR
END_METHOD

END_FUNCTION_BLOCK

// ---- POUs/Classes/ROBOT_DATA_HANDLER.TcPOU
FUNCTION_BLOCK ROBOT_DATA_HANDLER
VAR_INPUT
END_VAR
VAR_OUTPUT
END_VAR
VAR
	
END_VAR

METHOD PUBLIC DATA_TO_STRING : STRING
VAR_INPUT
END_VAR
VAR
	emptyJointsString : STRING := '0.0 0.0 0.0 0.0 0.0';
	separator : STRING := ' ';
	
	debugValue : LREAL := 10.0;
END_VAR
// CONVERT MOVEMENT DATA TO ROBOT MOVEMENT STRING.

//GVL.robotData.joint0.speed := 0.0; // DEBUG REMOVE LATER
//GVL.robotData.joint1.speed := 0.0; // DEBUG REMOVE LATER
//GVL.robotData.joint2.speed := 0.0; // DEBUG REMOVE LATER
//GVL.robotData.joint3.speed := 0.0; // DEBUG REMOVE LATER

DATA_TO_STRING :=
	CONCAT(LREAL_TO_STRING(GVL.robotData.joint0.curSpeed), 
	CONCAT(separator, 
	CONCAT(LREAL_TO_STRING(GVL.robotData.joint1.curSpeed),
	CONCAT(separator, 
	CONCAT(LREAL_TO_STRING(GVL.robotData.joint2.curSpeed),
	CONCAT(separator,  
	CONCAT(LREAL_TO_STRING(GVL.robotData.joint3.curSpeed),
	CONCAT(separator,
		emptyJointsString))))))));
END_METHOD

METHOD PUBLIC DEGREES_TO_MOVEMENT_DATA : BOOL
VAR_INPUT
	degrees : LREAL;
	jointNr : INT;
END_VAR
VAR
	moveTime : TIME;
	moveSpeed : LREAL;
	tempTimeValue : LREAL;
	speedMultiplier : LREAL := 3;
	TimePerDegree : LREAL := 544;
	TimePerDegree3 : LREAL := 390;
	tempDegrees : LREAL;
END_VAR
CASE jointNr OF
	0:
		tempDegrees := degrees - GVL.robotData.joint0.curPosition;
	1:
		tempDegrees := degrees - GVL.robotData.joint1.curPosition;
	2:
		tempDegrees := degrees - GVL.robotData.joint2.curPosition;
	3:
		tempDegrees := degrees - GVL.robotData.joint3.curPosition;
END_CASE

IF (tempDegrees < 0) THEN
	moveSpeed := 20.0;
	tempDegrees := tempDegrees * -1;
ELSIF (tempDegrees > 0) THEN
	moveSpeed := -20.0;
	tempDegrees := tempDegrees;
END_IF


moveSpeed := moveSpeed * speedMultiplier;
IF (jointNr = 3) THEN
	tempTimeValue := ((tempDegrees * TimePerDegree3) / speedMultiplier);
ELSE
	tempTimeValue := ((tempDegrees * TimePerDegree) / speedMultiplier);
END_IF
moveTime := LREAL_TO_TIME(tempTimeValue);


CASE jointNr OF
	0:
		GVL.robotData.joint0.timer.timerTime := moveTime;
		GVL.robotData.joint0.setSpeed := moveSpeed;
		GVL.robotData.joint0.curPosition := degrees;
	1:
		GVL.robotData.joint1.timer.timerTime := moveTime;
		GVL.robotData.joint1.setSpeed := moveSpeed;
		GVL.robotData.joint1.curPosition := degrees;
	2:
		GVL.robotData.joint2.timer.timerTime := moveTime;
		GVL.robotData.joint2.setSpeed := moveSpeed;
		GVL.robotData.joint2.curPosition := degrees;
	3:
		GVL.robotData.joint3.timer.timerTime := moveTime;
		GVL.robotData.joint3.setSpeed := moveSpeed;
		GVL.robotData.joint3.curPosition := degrees;
END_CASE
END_METHOD

METHOD PUBLIC JOINT_DATA_HANDLER : BOOL
VAR_INPUT
END_VAR
// TURN RECEIVED ROBOT DATA INTO CURRENT JOINTS POSITIONS
// DONT USE THIS METHOD!!!!!!!!!!

IF (GVL.ReceivedStringArray[0] = 'CRISTART') THEN
	// WHAT IS THE LOCATION
END_IF


// WE CAN'T GET THE CURRENT LOCATION FROM THE ROBOT SO WE LEFT THIS EMPTY FOR NOW!!
END_METHOD

METHOD PUBLIC MOVEMENT_CONTROLLER : BOOL
VAR_INPUT
END_VAR
VAR
	count : INT := 0;
END_VAR
//Base
IF (GVL.robotData.joint0.setSpeed <> 0 AND GVL.robotData.isBusy[4] = FALSE) THEN
	GVL.robotData.joint0.timer.timerStart := TRUE;
	GVL.robotData.joint0.curSpeed := GVL.robotData.joint0.setSpeed;
	GVL.robotData.joint0.setSpeed := 0;
	GVL.robotData.isBusy[0] := TRUE;
ELSIF(GVL.robotData.joint0.timer.timerCon.Q) THEN
	GVL.robotData.joint0.timer.timerStart := FALSE;
	GVL.robotData.joint0.curSpeed := 0.0;
	GVL.robotData.isBusy[0] := FALSE;
END_IF

//Arm 1
IF (GVL.robotData.joint1.setSpeed <> 0 AND GVL.robotData.isBusy[4] = FALSE) THEN
	GVL.robotData.joint1.timer.timerStart := TRUE;
	GVL.robotData.joint1.curSpeed := GVL.robotData.joint1.setSpeed;
	GVL.robotData.joint1.setSpeed := 0;
	GVL.robotData.isBusy[1] := TRUE;
ELSIF(GVL.robotData.joint1.timer.timerCon.Q) THEN
	GVL.robotData.joint1.timer.timerStart := FALSE;
	GVL.robotData.joint1.curSpeed := 0.0;
	GVL.robotData.isBusy[1] := FALSE;
END_IF

//Arm2
IF (GVL.robotData.joint2.setSpeed <> 0 AND GVL.robotData.isBusy[4] = FALSE) THEN
	GVL.robotData.joint2.timer.timerStart := TRUE;
	GVL.robotData.joint2.curSpeed := GVL.robotData.joint2.setSpeed;
	GVL.robotData.joint2.setSpeed := 0;
	GVL.robotData.isBusy[2] := TRUE;
ELSIF(GVL.robotData.joint2.timer.timerCon.Q) THEN
	GVL.robotData.joint2.timer.timerStart := FALSE;
	GVL.robotData.joint2.curSpeed := 0.0;
	GVL.robotData.isBusy[2] := FALSE;
END_IF

//Arm3
IF (GVL.robotData.joint3.setSpeed <> 0 AND GVL.robotData.isBusy[4] = FALSE) THEN
	GVL.robotData.joint3.timer.timerStart := TRUE;
	GVL.robotData.joint3.curSpeed := GVL.robotData.joint3.setSpeed;
	GVL.robotData.joint3.setSpeed := 0;
	GVL.robotData.isBusy[3] := TRUE;
ELSIF(GVL.robotData.joint3.timer.timerCon.Q) THEN
	GVL.robotData.joint3.timer.timerStart := FALSE;
	GVL.robotData.joint3.curSpeed := 0.0;
	GVL.robotData.isBusy[3] := FALSE;
END_IF

//Global busy indicator
IF (GVL.robotData.isBusy[0] = FALSE AND GVL.robotData.isBusy[1] = FALSE AND GVL.robotData.isBusy[2] = FALSE AND GVL.robotData.isBusy[3] = FALSE) THEN
	GVL.robotData.isBusy[4] := FALSE;
ELSE
	GVL.robotData.isBusy[4] := TRUE;
END_IF
END_METHOD

METHOD PUBLIC SET_JOINTS_TO_POSITION : BOOL
VAR_INPUT
	X : LREAL;
	Z : LREAL;
	Y : LREAL;
	baseOffsetDegrees : LREAL := 0;	//Positive numbers = right, negative numbers left
END_VAR
VAR
	baseRotation : LREAL;
	actualBaseRotation : LREAL;
	arm1Rotation : LREAL;
	arm2Rotation : LREAL;
	arm3Rotation : LREAL;
	targetPosition : Position;
	
END_VAR
targetPosition.x := X;
targetPosition.z := Z;
targetPosition.y := Y;

TARGET_TO_DEGREES_CALCULATOR(targetPosition, baseDegrees => baseRotation, 
										     arm1Degrees => arm1Rotation,
											 arm2Degrees => arm2Rotation,
											 arm3Degrees => arm3Rotation);

actualBaseRotation := baseRotation + baseOffsetDegrees;

IF (actualBaseRotation > GVL_RobotArmConstants.MAXIMUM_BASE_ROTATION_FROM_CENTER) THEN
	//Cap right
	actualBaseRotation := GVL_RobotArmConstants.MAXIMUM_BASE_ROTATION_FROM_CENTER;
ELSIF (actualBaseRotation < (-1.0 * GVL_RobotArmConstants.MAXIMUM_BASE_ROTATION_FROM_CENTER)) THEN
	//Cap left
	actualBaseRotation := -1.0 * GVL_RobotArmConstants.MAXIMUM_BASE_ROTATION_FROM_CENTER;
END_IF

//Set all joints to calcualted angles
DEGREES_TO_MOVEMENT_DATA(jointNr := 0, degrees := actualBaseRotation);
DEGREES_TO_MOVEMENT_DATA(jointNr := 1, degrees := arm1Rotation);						 
DEGREES_TO_MOVEMENT_DATA(jointNr := 2, degrees := arm2Rotation);
DEGREES_TO_MOVEMENT_DATA(jointNr := 3, degrees := arm3Rotation);
END_METHOD

METHOD PUBLIC TARGET_TO_DEGREES_CALCULATOR : BOOL
VAR_INPUT
	targetPosition : Position;
END_VAR
VAR_OUTPUT
	baseDegrees : LREAL;
	arm1Degrees : LREAL;
	arm2Degrees : LREAL;
	arm3Degrees : LREAL;
END_VAR
// TURN CURRENT POSITION AND TARGET POSITION TO INTO MOVEMENT PER JOINT.
baseDegrees := GetBaseAngleDegrees(targetPosition);
GetArm1AndArm2Degrees(position := targetPosition, arm1Degrees => arm1Degrees, arm2Degrees => arm2Degrees);
arm3Degrees := GetArm3RotationPerpendicularToGround(arm1Degrees, arm2Degrees);
END_METHOD

METHOD PUBLIC TO_ZERO : BOOL
VAR_INPUT
END_VAR
DEGREES_TO_MOVEMENT_DATA(degrees := 0, jointNr := 0);
DEGREES_TO_MOVEMENT_DATA(degrees := 0, jointNr := 1);
DEGREES_TO_MOVEMENT_DATA(degrees := 0, jointNr := 2);
DEGREES_TO_MOVEMENT_DATA(degrees := 0, jointNr := 3);
END_METHOD

END_FUNCTION_BLOCK

// ---- POUs/InverseKinematics/GetBaseAngleDegrees.TcPOU
/// Gets the angle to which the base has to rotate. 
/// Negative value to rotate left, positive value to rotate right
FUNCTION GetBaseAngleDegrees : LREAL
VAR_INPUT
	position : Position;	//The target position
END_VAR
VAR
	xSide : LREAL;
	halfAreaWidth : LREAL;
	zSide : LREAL;
	angleOffset : LREAL := 1.0;
	targetAngleDegrees : LREAL;
END_VAR

xSide := GVL_RobotArmConstants.DISTANCE_TO_PICKUP_AREA + position.x;
halfAreaWidth := GVL_RobotArmConstants.PICKUP_AREA_WIDTH / 2;

IF (position.z < halfAreaWidth) THEN
	zSide := halfAreaWidth - position.z;
	angleOffset := -1.0;
ELSE
	zSide := position.z - halfAreaWidth;
	angleOffset := 1.0;
END_IF

targetAngleDegrees := GetAngleDegreesFromOppositeAndAdjacent(opposite := zSide, adjacent := xSide);
GetBaseAngleDegrees := targetAngleDegrees * angleOffset;

END_FUNCTION

// ---- POUs/InverseKinematics/GetAngleDegreesFromOppositeAndAdjacent.TcPOU
/// Calculates an angle in a right triangle based on the 2 non-hypotenuse sides
/// Returns the angle, in degrees
FUNCTION GetAngleDegreesFromOppositeAndAdjacent : LREAL
VAR_INPUT
	opposite : LREAL; //the side opposite the angle
	adjacent : LREAL; //the side next to the angle (not hypotenuse)
END_VAR
VAR
	tangentFraction : LREAL;
	targetAngleRadians : LREAL;
	targetAngleDegrees : LREAL;
END_VAR

tangentFraction := opposite / adjacent;
targetAngleRadians := ATAN(tangentFraction); //No need to worry about which quadrant we are in, as we are working with a right-angle triangle so we can only be in the first one
targetAngleDegrees := RadiansToDegrees(targetAngleRadians);

GetAngleDegreesFromOppositeAndAdjacent := targetAngleDegrees;

END_FUNCTION

// ---- POUs/InverseKinematics/RadiansToDegrees.TcPOU
FUNCTION RadiansToDegrees : LREAL
VAR_INPUT
	radians : LREAL;
END_VAR
VAR
END_VAR

RadiansToDegrees := radians * 180 / GVL_RobotArmConstants.Pi;

END_FUNCTION

// ---- POUs/InverseKinematics/GetArm1AndArm2Degrees.TcPOU
FUNCTION GetArm1AndArm2Degrees : BOOL
VAR_INPUT
	position : Position;
END_VAR
VAR_OUTPUT
	arm1Degrees : LREAL;
	arm2Degrees : LREAL;
END_VAR
VAR
	actualY : LREAL;
	
	oppositeSide : LREAL;
	adjacentSide : LREAL;
	baseTriangleHypotenuse : LREAL;
	angleDegreesFromBaseToActualY : LREAL;
	
	armTriangleBase : LREAL;
	armTriangleA : LREAL;
	armTriangleB : LREAL;
	
	arm1AngleDegreesRelativeToBaseTriangle : LREAL;
	arm2DegreesRelativeArm1 : LREAL;
END_VAR

actualY := position.y - GVL_RobotArmConstants.ARM_BASE_HEIGHT + GVL_RobotArmConstants.ARM_3_LENGTH + GVL_RobotArmConstants.GRABBER_HEIGHT;

IF (actualY < 0) THEN
	arm1Degrees := 0;
	arm2Degrees := 0;
	GetArm1AndArm2Degrees := FALSE;
	RETURN;
END_IF

oppositeSide := actualY;
adjacentSide := GetDistanceToPositionFromBase2D(position);
baseTriangleHypotenuse := GetHypotenuse(oppositeSide, adjacentSide);
angleDegreesFrombaseToActualY := GetAngleDegreesFromOppositeAndAdjacent(oppositeSide, adjacentSide);

armTriangleBase := baseTriangleHypotenuse;
armTriangleA := GVL_RobotArmConstants.ARM_1_LENGTH;
armTriangleB := GVL_RobotArmConstants.ARM_2_LENGTH;

arm1AngleDegreesRelativeToBaseTriangle := GetAngleDegreesFrom3Sides(armTriangleA, armTriangleB, armTriangleBase);
arm1Degrees := (angleDegreesFromBaseToActualY + arm1AngleDegreesRelativeToBaseTriangle) - 90;

arm2DegreesRelativeArm1 := GetAngleDegreesFrom3Sides(armTriangleB, armTriangleBase, armTriangleA);
arm2Degrees := arm2DegreesRelativeArm1 - 90;

END_FUNCTION

// ---- POUs/InverseKinematics/GetDistanceToPositionFromBase2D.TcPOU
FUNCTION GetDistanceToPositionFromBase2D : LREAL
VAR_INPUT
	position : Position;	//The target position
END_VAR
VAR
	xSide : LREAL;
	zSide : LREAL;
END_VAR

xSide := GetXSide(position.x);
zSide := GetZSide(position.z);

GetDistanceToPositionFromBase2D := GetHypotenuse(xSide, zSide);

END_FUNCTION

// ---- POUs/InverseKinematics/GetXSide.TcPOU
FUNCTION GetXSide : LREAL
VAR_INPUT
	xPos : LREAL;
END_VAR
VAR
END_VAR

GetXSide := GVL_RobotArmConstants.DISTANCE_TO_PICKUP_AREA + xPos;

END_FUNCTION

// ---- POUs/InverseKinematics/GetZSide.TcPOU
FUNCTION GetZSide : LREAL
VAR_INPUT
	zPos : LREAL;
END_VAR
VAR
	zSide : LREAL;
	halfAreaWidth : LREAL;
END_VAR

halfAreaWidth := GVL_RobotArmConstants.PICKUP_AREA_WIDTH / 2;

IF (zPos < halfAreaWidth) THEN
	//Point is on the left side of the robot
	zSide := halfAreaWidth - zPos;
ELSE
	//Point is on the right side of the robot
	zSide := zPos - halfAreaWidth;
END_IF

GetZSide := zSide;

END_FUNCTION

// ---- POUs/InverseKinematics/GetHypotenuse.TcPOU
FUNCTION GetHypotenuse : LREAL
VAR_INPUT
	a : LREAL;
	b : LREAL;
END_VAR
VAR
	resultSquared : LREAL;
END_VAR

resultSquared := a * a + b * b;
GetHypotenuse := SQRT(resultSquared);

END_FUNCTION

// ---- POUs/InverseKinematics/GetAngleDegreesFrom3Sides.TcPOU
FUNCTION GetAngleDegreesFrom3Sides : LREAL
VAR_INPUT
	adjacentLeft : LREAL;
	opposite : LREAL;
	adjacentRight : LREAL;
END_VAR
VAR
	cosTargetAngle : LREAL;
	targetAngleRadians : LREAL;
END_VAR

//Cosine formula
cosTargetAngle := ((adjacentLeft * adjacentLeft) + (adjacentRight * adjacentRight) - (opposite * opposite))
				  /
				  (2 * adjacentLeft * adjacentRight);
				  
targetAngleRadians := ACOS(cosTargetAngle);

GetAngleDegreesFrom3Sides := RadiansToDegrees(targetAngleRadians);

END_FUNCTION

// ---- POUs/InverseKinematics/GetArm3RotationPerpendicularToGround.TcPOU
FUNCTION GetArm3RotationPerpendicularToGround : LREAL
VAR_INPUT
	arm1RotationDegrees : LREAL;
	arm2RotationDegrees : LREAL;
END_VAR
VAR
END_VAR

GetArm3RotationPerpendicularToGround := -1.0 * (arm1RotationDegrees + arm2RotationDegrees);

END_FUNCTION

// ---- POUs/Classes/ArmMovementHandler.TcPOU
FUNCTION_BLOCK ArmMovementHandler
VAR_INPUT
END_VAR
VAR_OUTPUT
END_VAR
VAR
	m_robotDataHandler : REFERENCE TO ROBOT_DATA_HANDLER;
	m_prevMovementState : ArmMovementState := ArmMovementState.NONE;
	m_currentMovementState : ArmMovementState := ArmMovementState.IDLE;
	
	m_objectInteractionTimer : TON;	//Timer to stay at the pickup/dropoff point
	m_isInteractionTimerOn : BOOL := FALSE;
	m_objectInteractionTime : TIME := T#5S;
	
	m_currentTargetPosition : Position;
END_VAR

//Always run
//Timers
GVL.robotData.joint0.timer.timerCon(IN := GVL.robotData.joint0.timer.timerStart, PT := GVL.robotData.joint0.timer.timerTime);
GVL.robotData.joint1.timer.timerCon(IN := GVL.robotData.joint1.timer.timerStart, PT := GVL.robotData.joint1.timer.timerTime);
GVL.robotData.joint2.timer.timerCon(IN := GVL.robotData.joint2.timer.timerStart, PT := GVL.robotData.joint2.timer.timerTime);
GVL.robotData.joint3.timer.timerCon(IN := GVL.robotData.joint3.timer.timerStart, PT := GVL.robotData.joint3.timer.timerTime);

m_robotDataHandler.MOVEMENT_CONTROLLER();

m_objectInteractionTimer(IN := m_isInteractionTimerOn, PT := m_objectInteractionTime);

CASE m_currentMovementState OF
	ArmMovementState.IDLE:
		IF (m_prevMovementState <> m_currentMovementState) THEN
			//Set target to default
			m_robotDataHandler.TO_ZERO();
			m_robotDataHandler.MOVEMENT_CONTROLLER();	//Put into all on-entry code to ensure the isBusy variables are properly updated
		END_IF
		
		m_prevMovementState := m_currentMovementState;
		m_currentMovementState := HandleIdleState();
		
		IF (m_prevMovementState <> m_currentMovementState) THEN
			//on exit code
		END_IF
	
	//
	ArmMovementState.PICKING:
		IF (m_prevMovementState <> m_currentMovementState) THEN
			//on-entry code
			//Target position acquired by remote
			m_robotDataHandler.SET_JOINTS_TO_POSITION(X := GVL.robotData.targetX, 
													  Z := GVL.robotData.targetZ,
													  Y := GVL.robotData.targetY,
													  baseOffsetDegrees := 0);
			m_robotDataHandler.MOVEMENT_CONTROLLER();
			GVL.robotData.isAtDefaultPosition := FALSE;
		END_IF
		m_prevMovementState := m_currentMovementState;
		m_currentMovementState := HandlePickingState();
		
		IF (m_prevMovementState <> m_currentMovementState) THEN
			//on exit code
			GVL.robotData.hasNewData := FALSE;
		END_IF
	//
	ArmMovementState.DROPPING:
		IF (m_prevMovementState <> m_currentMovementState) THEN
			//on-entry code
			m_robotDataHandler.SET_JOINTS_TO_POSITION(X := GVL_RobotArmConstants.DROPOFF_X, 
													  Z := GVL_RobotArmConstants.DROPOFF_Z,
													  Y := GVL.robotData.targetY,
													  baseOffsetDegrees := GVL_RobotArmConstants.DROPOFF_BASE_OFFSET);
			GVL.robotData.isAtDefaultPosition := FALSE;
			m_robotDataHandler.MOVEMENT_CONTROLLER();
		END_IF
		m_prevMovementState := m_currentMovementState;
		m_currentMovementState := HandleDroppingState();
		
		IF (m_prevMovementState <> m_currentMovementState) THEN
			//on exit code
		END_IF
	//
END_CASE

METHOD PUBLIC BindRobotDataHandler : BOOL
VAR_INPUT
	dataHandler : REFERENCE TO ROBOT_DATA_HANDLER;
END_VAR
m_robotDataHandler REF= dataHandler;
END_METHOD

METHOD PRIVATE HandleDroppingState : ArmMovementState
VAR_INPUT
END_VAR
HandleDroppingState := ArmMovementState.DROPPING;

IF (GVL.robotData.isBusy[4]) THEN
	RETURN;
END_IF

//Dropoff reached
m_isInteractionTimerOn := TRUE;

IF (m_objectInteractionTimer.Q) THEN
	//We have waited enough
	m_isInteractionTimerOn := FALSE;
	HandleDroppingState := ArmMovementState.IDLE;
END_IF
END_METHOD

METHOD PRIVATE HandleIdleState : ArmMovementState
VAR_INPUT
END_VAR
HandleIdleState := ArmMovementState.IDLE;

IF (GVL.robotData.isBusy[4]) THEN
	RETURN;
END_IF

//Not busy anymore
GVL.robotData.isAtDefaultPosition := TRUE;

IF (GVL.robotData.hasNewData) THEN
	HandleIdleState := ArmMovementState.PICKING;
END_IF
END_METHOD

METHOD PRIVATE HandlePickingState : ArmMovementState
VAR_INPUT
END_VAR
HandlePickingState := ArmMovementState.PICKING;

// 
IF (GVL.robotData.isBusy[4]) THEN
	RETURN;
END_IF

//We are at the picking destination
m_isInteractionTimerOn := TRUE;

IF (m_objectInteractionTimer.Q) THEN
	//We have waited enough
	m_isInteractionTimerOn := FALSE;
	HandlePickingState := ArmMovementState.DROPPING;
END_IF
END_METHOD

END_FUNCTION_BLOCK

// ---- POUs/Helpers/ShiftHistoryLeft.TcPOU
FUNCTION ShiftHistoryLeft : BOOL
VAR_INPUT
	//TODO: Use constant in GVL_Constants
	arr : REFERENCE TO ARRAY[0..9] OF MessageLogData;
END_VAR
VAR
	i : INT := 0;
END_VAR

FOR i:= 0 TO 9 - 1 BY 1 DO
	arr[i] := arr[i + 1];
END_FOR

END_FUNCTION

// ---- POUs/Helpers/AddCounterToMessage.TcPOU
FUNCTION AddCounterToMessage : T_MaxString
VAR_INPUT
	counter : INT;
	message : T_MaxString;
END_VAR
VAR
END_VAR

AddCounterToMessage := CONCAT('CRISTART ', 
					   CONCAT(INT_TO_STRING(counter), 
					   CONCAT(' ',
					   CONCAT(message, 
							 ' CRIEND'))));

END_FUNCTION

// ---- GlobalTextList.TcGTLO
TEXTLIST GlobalTextList
  423 = 'Connect'
  286 = 'Connect To Robot'
  403 = 'Debug Send'
  411 = 'Disable Motors'
  428 = 'Disconnect'
  622 = 'Enable Motors'
  229 = 'History'
  576 = 'Joint : '
  308 = 'Joint0 : '
  296 = 'Joint1 : '
  504 = 'Joint2 : '
  56 = 'Joint3 : '
  770 = 'Left'
  290 = 'Message'
  597 = 'Messages received: %d'
  193 = 'Receive History'
  495 = 'Reset'
  93 = 'Right'
  729 = 'Send'
  247 = 'Send / Send Command'
  222 = 'Server: %s'
  529 = 'Status: %s'
  75 = 'Stop'
  256 = 'Time'
  297 = 'To Idle Position'
  615 = 'To Idle Position / Send '
  485 = 'To Idle Position / Send Var'
END_TEXTLIST

// ---- VISUs/VisualizationControlPanel.TcVIS
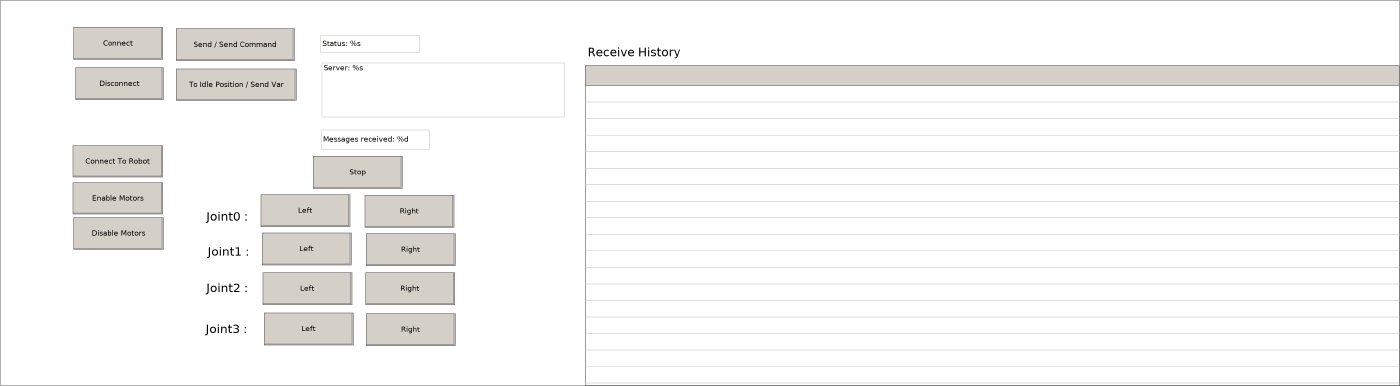
VISUALIZATION VisualizationControlPanel  // 2116x584
    Button (114,102 133x49), "Disconnect"
        tap MAIN.buttonDisconnectPressed
    Button (266,43 179x49), "Send / Send Command"
        tap MAIN.buttonSendPressed
    Button (111,41 135x49), "Connect"
        tap MAIN.buttonConnectPressed
    Textfield (486,95 367x82), "Server: %s", text variable: MAIN.messageFromServer
    Textfield (485,196 164x30), "Messages received: %d", text variable: MAIN.totalMessagesFromServerCount
    Table (884,99 1232x485), data array: MAIN.messageHistoryArray
        p3854506369: MAIN.messageHistoryArray[INDEX].systemTimeString
        p1892666644: MAIN.messageHistoryArray[INDEX].message
        p511219082: Message
    Label (885,64 182x30), "Receive History"
    Button (110,220 136x48), "Connect To Robot"
        tap MAIN.buttonConnectToRobotPressed
    Button (266,104 182x48), "To Idle Position / Send Var"
        tap MAIN.buttonDebugSendPressed
    Button (110,276 136x48), "Enable Motors"
        tap MAIN.buttonEnableMotorsPressed
    Textfield (484,53 150x26), "Status: %s", text variable: MAIN.connectionMessage
    Button (111,329 136x48), "Disable Motors"
        tap MAIN.buttonDisableMotorsPressed
    Button (394,294 135x49), "Left"
        tap MAIN.buttonLeft0Pressed
    Button (551,295 135x49), "Right"
        tap MAIN.buttonRight0Pressed
    Button (473,236 135x49), "Stop"
        tap MAIN.buttonStopPressed
    Label (311,366 90x30), "Joint1 :"
    Button (553,353 135x49), "Right"
        tap MAIN.buttonRight1Pressed
    Button (552,412 135x49), "Right"
        tap MAIN.buttonRight2Pressed
    Button (553,474 135x49), "Right"
        tap MAIN.buttonRight3Pressed
    Button (396,352 135x49), "Left"
        tap MAIN.buttonLeft1Pressed
    Button (397,412 135x49), "Left"
        tap MAIN.buttonLeft2Pressed
    Button (399,473 135x49), "Left"
        tap MAIN.buttonLeft3Pressed
    Label (309,313 90x30), "Joint0 :"
    Label (309,421 90x30), "Joint2 :"
    Label (308,483 90x30), "Joint3 :"
END_VISUALIZATION
